Omron CX-Programmer project NewProject (CX-Programmer 9.51)

# PLC Assignment1: CP1L-E EL

## Global symbols (name address type ; comment)
1000 CHANNEL  ; O_W_E_T_Interval
T0011 BOOL  ; SRH_300

## Program NewProgram1 (cyclic task 0)
Local symbols
Arm_extends 100.05 BOOL
Arm_retracts 100.06 BOOL
Boot_Finish 2.08 BOOL  ; Has booted up
Bootup_Interval 50 NUMBER  ; Boot up for 5s
Bootup_Timer 1 NUMBER  ; Timer for bootup period
Bootup_Timer_Done T0001 BOOL  ; RUN Bootup Timer
ConvB_In_Timer 9 NUMBER  ; Timer for Conv B In
ConvB_In_Timer_Done T0009 BOOL  ; ConvB in stops
ConvB_Interval 100 NUMBER  ; ConvB stops for 10s
ConvB_Out_Interval 10.00 BOOL  ; sending pallet out for 10s
ConvB_Out_Timer 10 NUMBER  ; Timer for conv B out
ConvB_Out_Timer_Done T0010 BOOL  ; ConvB moving out timer
Converyor_B_IN 100.01 BOOL
Conveyor_A_on 100.00 BOOL
Conveyor_B_OUT 100.02 BOOL
Cycle_Count_Done C0001 BOOL  ; Cycle Counter
END_light 100.07 BOOL
EW_Mode 1.08 BOOL  ; Extend to Grab Widget Mode
End_Light_Flash_Interval 10 NUMBER  ; Flash for 1s
First_Widget 2.09 BOOL  ; if it is first widget placed
Flash_Timer1_Done T0015 BOOL  ; End Light flash 1s Timer1 ends
Flash_Timer2_Done T0016 BOOL  ; End light flash 1s Timer2 ends
GW_Interval 10 NUMBER  ; grab widget for 1s
GW_Mode 1.07 BOOL  ; Grab Widget Mode
GW_Timer 4 NUMBER  ; Timer for grab widget period
GW_Timer_Done T0004 BOOL  ; Grab Widget Timer
G_W_T_Done T0003 BOOL  ; Grip_Widget_Timer
G_W_T_Interval 50 NUMBER  ; grip widget for 5s
G_W_T_Timer 3 NUMBER  ; Timer for grip widget period
Has_Entered_Reset 2.12 BOOL  ; check if the machine has ever entered reset state
Has_Placed_Widget 2.02 BOOL  ; has placed a widet in place widget section
Has_Retract_Arm 2.05 BOOL  ; have succesfuuly retract arm to home position
LP_Mode 1.04 BOOL  ; Load pallet mode
LP_Mode_Finish 1.13 BOOL  ; load pallet mode has finished
LS1 0.03 BOOL  ; Limit Switch 1
LS2 0.04 BOOL  ; Limit Switch 2
LW_Mode 1.05 BOOL  ; Load Widget Mode
LW_Mode_Finish 1.14 BOOL  ; Load widget mode finish
MR_Interval 50 NUMBER  ; retract arm for 5s
MR_Timer 8 NUMBER  ; Timer for retract widget period
MR_Timer_Done T0008 BOOL  ; Retract After Grabbing Widget
MW_Mode 1.09 BOOL  ; Move widget mode
MW_Mode_Finish 2.01 BOOL  ; move widget mode finished
OW_Mode 1.06 BOOL  ; Obtain Widget Mode
OW_Mode_Finish 2.00 BOOL  ; Obtain Widget Mode Finished
O_W_E_T_Done T0002 BOOL  ; Obtain Widget Extend Timer
O_W_E_T_Interval 50 NUMBER  ; 5s timer
O_W_E_T_Timer 2 NUMBER  ; Timer for Obtain Widget Extend Period
Operator_present 0.07 BOOL  ; Operator present sensor
PW_Mode 1.10 BOOL  ; Place Widget Mode
PW_Mode_Finish 2.03 BOOL  ; Place Widget has finished
PW_Wait_5s T0011 BOOL  ; Forced Wait 5s according to Step 5
P_E_300_Done T0007 BOOL  ; Place Widget Extend 300 Timer
P_E_300_Interval 30 NUMBER  ; extends arm 300mm for 3s
P_E_300_Timer 7 NUMBER  ; Timer for place widget extend 300mm period
P_E_400_Done T0006 BOOL  ; Place Widget Extend 400 Timer
P_E_400_Interval 40 NUMBER  ; extends arm 400mm for 4s
P_E_400_Timer 6 NUMBER  ; Timer for place widget extend 400mm period
P_E_500_Done T0005 BOOL  ; Place Widget Extend 500 Timer
P_E_500_Interval 50 NUMBER  ; extends arm 500mm for 5s
P_E_500_Timer 5 NUMBER  ; Timer for place widget extend 500mm period
Pallet_Detected 2.07 BOOL  ; Detect pallet in Load Pallet mode
Pallet_present 0.06 BOOL  ; Pallet present sensor
Power_On 0.08 BOOL
Reset 0.02 BOOL
Reset_Interval 50 NUMBER  ; Reset pressed 5s
Reset_Mode 1.02 BOOL
Reset_Timer 0 NUMBER  ; Timer for reset period
Reset_Timer_Done T0000 BOOL  ; Reset Pressed Timer
Run_Mode 1.00 BOOL
SCARA_anticlockwise 100.04 BOOL
SCARA_clockwise 100.03 BOOL
SP_Mode 1.12 BOOL  ; Send Pallet Mode
SP_Mode_Finish 1.15 BOOL  ; Send pallet out mode finish
SRH_Mode 1.11 BOOL  ; Scara Return Home
SRH_Mode_Finish 2.04 BOOL  ; Scara Return Home has finished
SRH_R_300 T0014 BOOL  ; Retract_Arm_2_Home_3s
SRH_R_400 T0013 BOOL  ; Retract_Arm_2_Home_4s
SRH_R_500 T0012 BOOL  ; Retract_Arm_2_Home_5s
Second_Widget 2.10 BOOL  ; If it is second widget placed
Standby_Mode 1.03 BOOL
Start 0.00 BOOL
Stop 0.01 BOOL
Stop_Mode 1.01 BOOL
Stop_Mode_Finish 2.13 BOOL  ; stopped everything
Third_Widget 2.11 BOOL  ; If it is third widget placed
Vision_part_present 0.05 BOOL
Widget_Count_Done C0000 BOOL  ; Widget Counter
Widget_Count_Num 3 NUMBER  ; Number of Widgets

### Section States_Transition

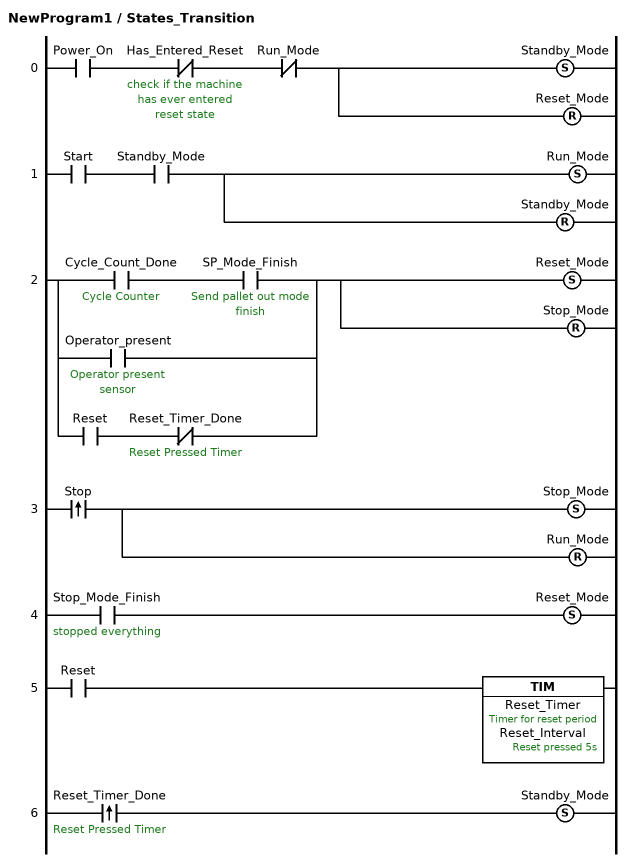
; rung 0
LD Power_On
ANDNOT Has_Entered_Reset  ; check if the machine has ever entered reset state
ANDNOT Run_Mode
SET Standby_Mode
RSET Reset_Mode
; rung 1
LD Start
AND Standby_Mode
SET Run_Mode
RSET Standby_Mode
; rung 2
LD Cycle_Count_Done  ; Cycle Counter
AND SP_Mode_Finish  ; Send pallet out mode finish
OR Operator_present  ; Operator present sensor
LD Reset
ANDNOT Reset_Timer_Done  ; Reset Pressed Timer
ORLD
SET Reset_Mode
RSET Stop_Mode
; rung 3
@LD Stop
SET Stop_Mode
RSET Run_Mode
; rung 4
LD Stop_Mode_Finish  ; stopped everything
SET Reset_Mode
; rung 5
LD Reset
TIM Reset_Timer Reset_Interval  ; Timer for reset period, Reset pressed 5s
; rung 6
@LD Reset_Timer_Done  ; Reset Pressed Timer
SET Standby_Mode

### Section Run

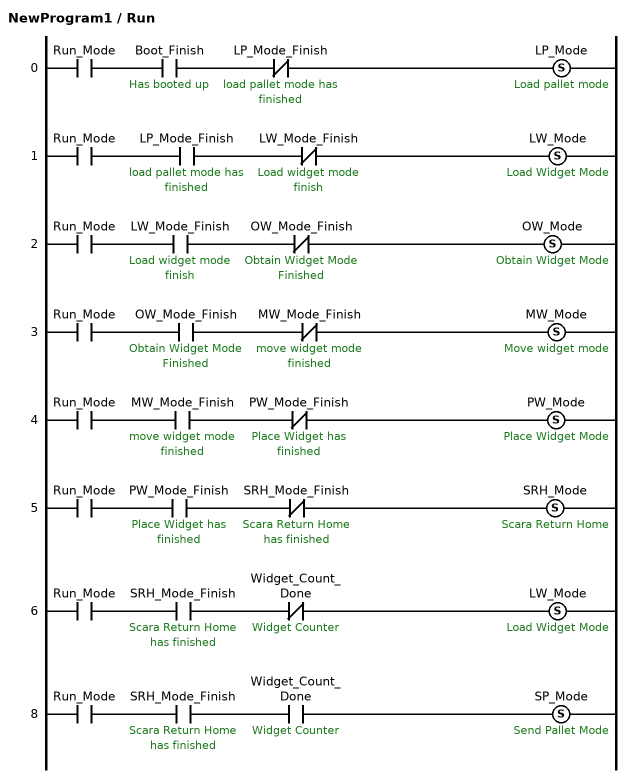
; rung 0
LD Run_Mode
AND Boot_Finish  ; Has booted up
ANDNOT LP_Mode_Finish  ; load pallet mode has finished
SET LP_Mode  ; Load pallet mode
; rung 1
LD Run_Mode
AND LP_Mode_Finish  ; load pallet mode has finished
ANDNOT LW_Mode_Finish  ; Load widget mode finish
SET LW_Mode  ; Load Widget Mode
; rung 2
LD Run_Mode
AND LW_Mode_Finish  ; Load widget mode finish
ANDNOT OW_Mode_Finish  ; Obtain Widget Mode Finished
SET OW_Mode  ; Obtain Widget Mode
; rung 3
LD Run_Mode
AND OW_Mode_Finish  ; Obtain Widget Mode Finished
ANDNOT MW_Mode_Finish  ; move widget mode finished
SET MW_Mode  ; Move widget mode
; rung 4
LD Run_Mode
AND MW_Mode_Finish  ; move widget mode finished
ANDNOT PW_Mode_Finish  ; Place Widget has finished
SET PW_Mode  ; Place Widget Mode
; rung 5
LD Run_Mode
AND PW_Mode_Finish  ; Place Widget has finished
ANDNOT SRH_Mode_Finish  ; Scara Return Home has finished
SET SRH_Mode  ; Scara Return Home
; rung 6
LD Run_Mode
AND SRH_Mode_Finish  ; Scara Return Home has finished
ANDNOT Widget_Count_Done  ; Widget Counter
SET LW_Mode  ; Load Widget Mode
; rung 8
LD Run_Mode
AND SRH_Mode_Finish  ; Scara Return Home has finished
AND Widget_Count_Done  ; Widget Counter
SET SP_Mode  ; Send Pallet Mode

### Section Stop

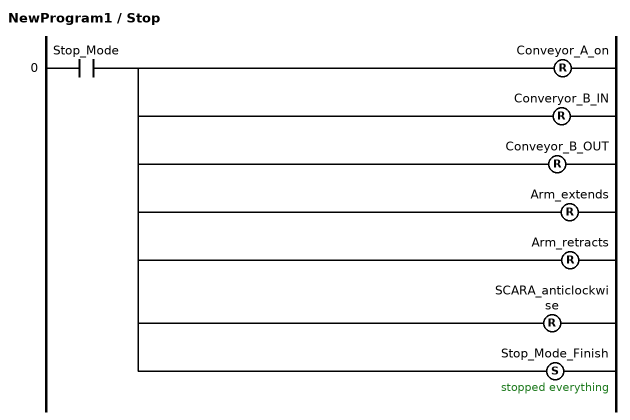
; rung 0
LD Stop_Mode
RSET Conveyor_A_on
RSET Converyor_B_IN
RSET Conveyor_B_OUT
RSET Arm_extends
RSET Arm_retracts
RSET SCARA_anticlockwise
SET Stop_Mode_Finish  ; stopped everything

### Section Reset

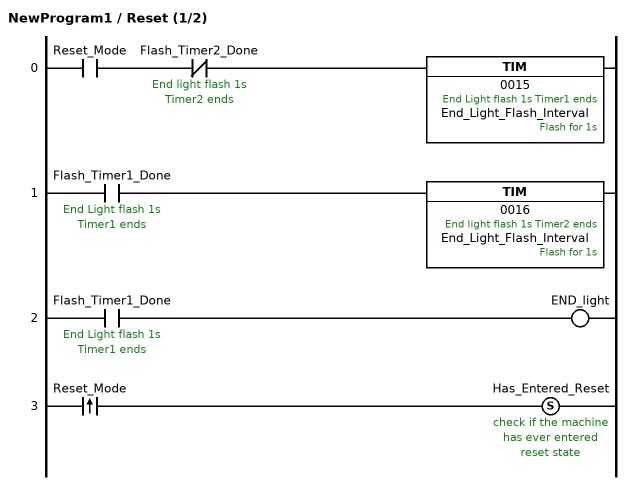
; rung 0
LD Reset_Mode
ANDNOT Flash_Timer2_Done  ; End light flash 1s Timer2 ends
TIM 0015 End_Light_Flash_Interval  ; Flash for 1s, End Light flash 1s Timer1 ends
; rung 1
LD Flash_Timer1_Done  ; End Light flash 1s Timer1 ends
TIM 0016 End_Light_Flash_Interval  ; Flash for 1s, End light flash 1s Timer2 ends
; rung 2
LD Flash_Timer1_Done  ; End Light flash 1s Timer1 ends
OUT END_light
; rung 3
@LD Reset_Mode
SET Has_Entered_Reset  ; check if the machine has ever entered reset state

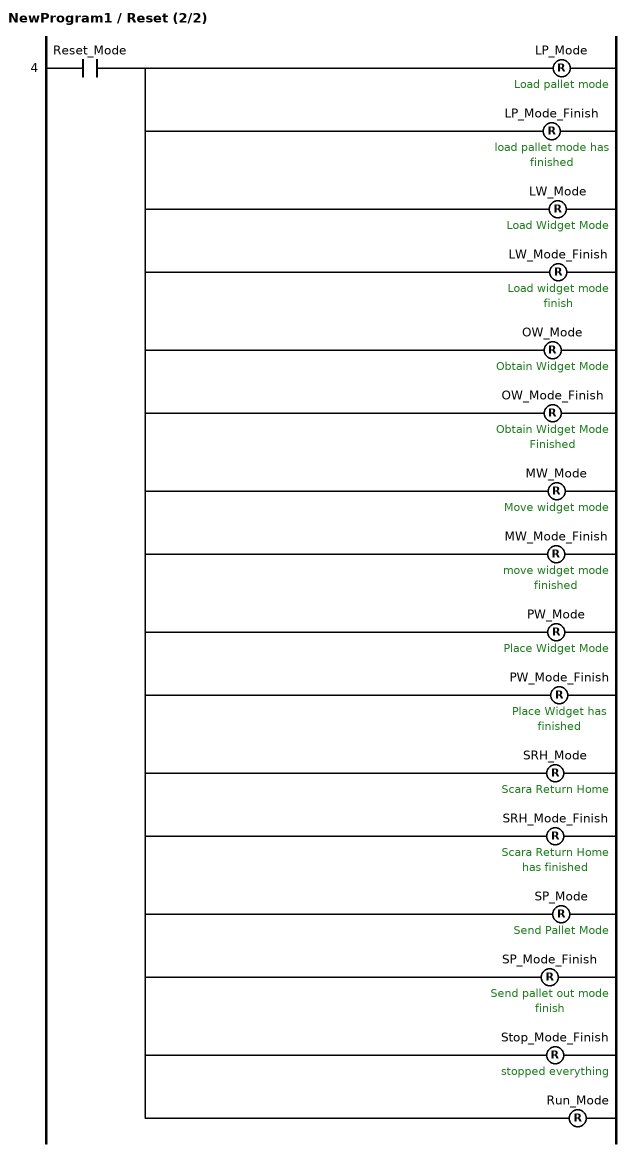
; rung 4
LD Reset_Mode
RSET LP_Mode  ; Load pallet mode
RSET LP_Mode_Finish  ; load pallet mode has finished
RSET LW_Mode  ; Load Widget Mode
RSET LW_Mode_Finish  ; Load widget mode finish
RSET OW_Mode  ; Obtain Widget Mode
RSET OW_Mode_Finish  ; Obtain Widget Mode Finished
RSET MW_Mode  ; Move widget mode
RSET MW_Mode_Finish  ; move widget mode finished
RSET PW_Mode  ; Place Widget Mode
RSET PW_Mode_Finish  ; Place Widget has finished
RSET SRH_Mode  ; Scara Return Home
RSET SRH_Mode_Finish  ; Scara Return Home has finished
RSET SP_Mode  ; Send Pallet Mode
RSET SP_Mode_Finish  ; Send pallet out mode finish
RSET Stop_Mode_Finish  ; stopped everything
RSET Run_Mode

### Section Standby

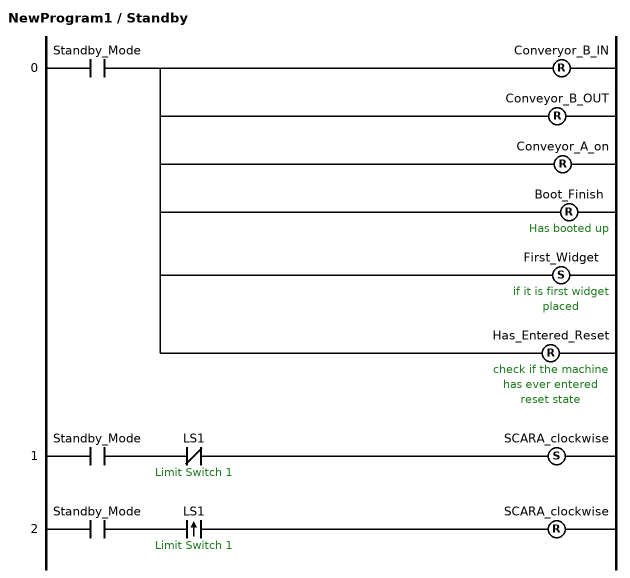
; rung 0
LD Standby_Mode
RSET Converyor_B_IN
RSET Conveyor_B_OUT
RSET Conveyor_A_on
RSET Boot_Finish  ; Has booted up
SET First_Widget  ; if it is first widget placed
RSET Has_Entered_Reset  ; check if the machine has ever entered reset state
; rung 1
LD Standby_Mode
ANDNOT LS1  ; Limit Switch 1
SET SCARA_clockwise
; rung 2
LD Standby_Mode
@AND LS1  ; Limit Switch 1
RSET SCARA_clockwise

### Section Boot_up

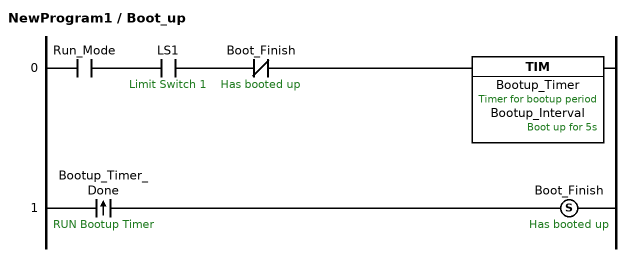
; rung 0
LD Run_Mode
AND LS1  ; Limit Switch 1
ANDNOT Boot_Finish  ; Has booted up
TIM Bootup_Timer Bootup_Interval  ; Timer for bootup period, Boot up for 5s
; rung 1
@LD Bootup_Timer_Done  ; RUN Bootup Timer
SET Boot_Finish  ; Has booted up

### Section LoadPallet

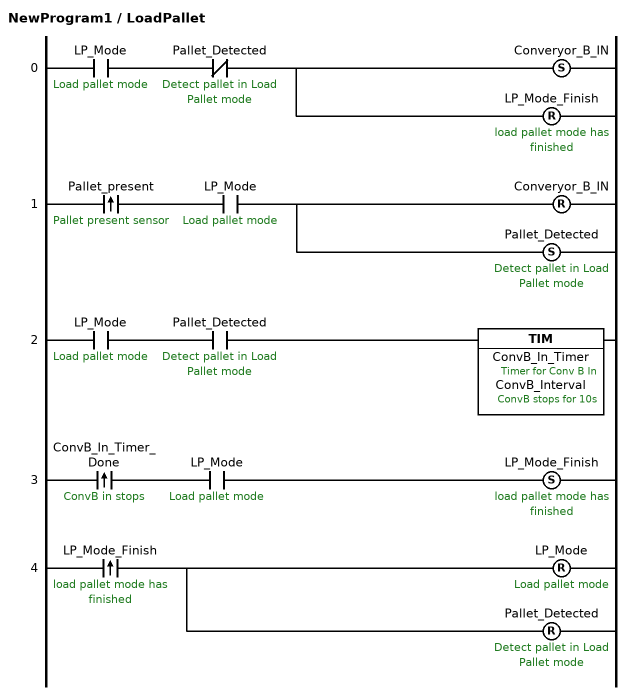
; rung 0
LD LP_Mode  ; Load pallet mode
ANDNOT Pallet_Detected  ; Detect pallet in Load Pallet mode
SET Converyor_B_IN
RSET LP_Mode_Finish  ; load pallet mode has finished
; rung 1
@LD Pallet_present  ; Pallet present sensor
AND LP_Mode  ; Load pallet mode
RSET Converyor_B_IN
SET Pallet_Detected  ; Detect pallet in Load Pallet mode
; rung 2
LD LP_Mode  ; Load pallet mode
AND Pallet_Detected  ; Detect pallet in Load Pallet mode
TIM ConvB_In_Timer ConvB_Interval  ; Timer for Conv B In, ConvB stops for 10s
; rung 3
@LD ConvB_In_Timer_Done  ; ConvB in stops
AND LP_Mode  ; Load pallet mode
SET LP_Mode_Finish  ; load pallet mode has finished
; rung 4
@LD LP_Mode_Finish  ; load pallet mode has finished
RSET LP_Mode  ; Load pallet mode
RSET Pallet_Detected  ; Detect pallet in Load Pallet mode

### Section LoadWidget

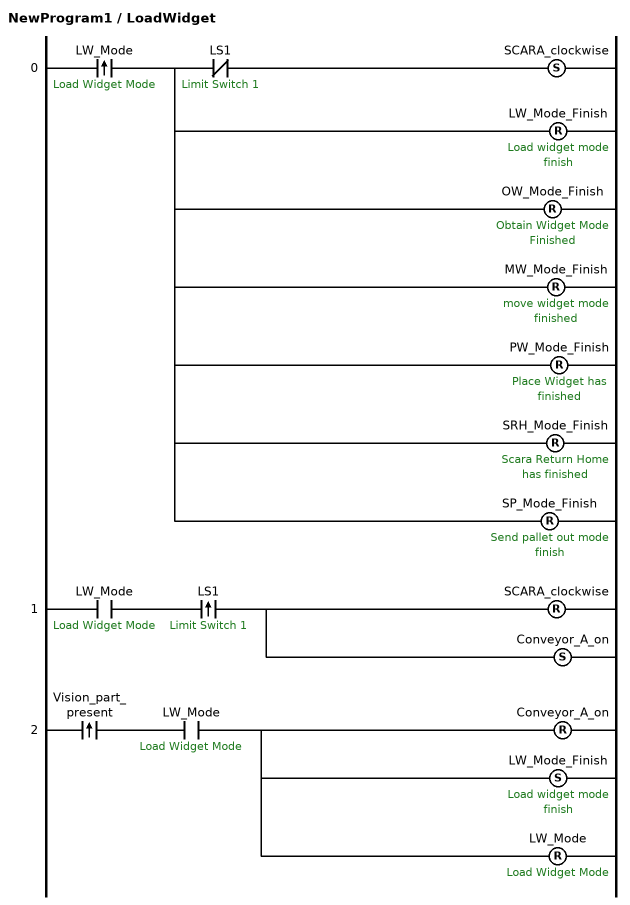
; rung 0
@LD LW_Mode  ; Load Widget Mode
OUT TR0
ANDNOT LS1  ; Limit Switch 1
SET SCARA_clockwise
LD TR0
RSET LW_Mode_Finish  ; Load widget mode finish
RSET OW_Mode_Finish  ; Obtain Widget Mode Finished
RSET MW_Mode_Finish  ; move widget mode finished
RSET PW_Mode_Finish  ; Place Widget has finished
RSET SRH_Mode_Finish  ; Scara Return Home has finished
RSET SP_Mode_Finish  ; Send pallet out mode finish
; rung 1
LD LW_Mode  ; Load Widget Mode
@AND LS1  ; Limit Switch 1
RSET SCARA_clockwise
SET Conveyor_A_on
; rung 2
@LD Vision_part_present
AND LW_Mode  ; Load Widget Mode
RSET Conveyor_A_on
SET LW_Mode_Finish  ; Load widget mode finish
RSET LW_Mode  ; Load Widget Mode

### Section ObtainWidget

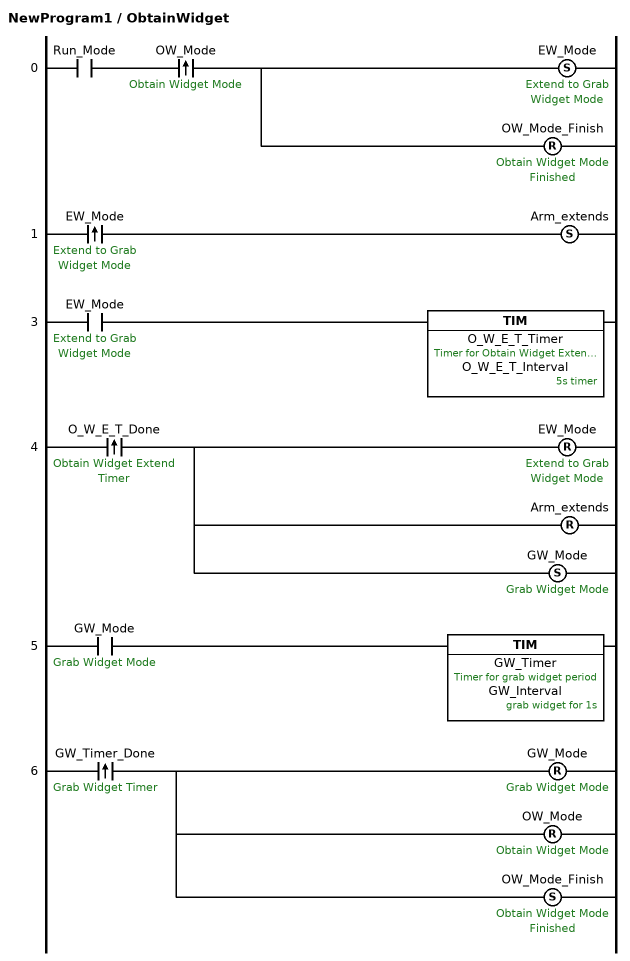
; rung 0
LD Run_Mode
@AND OW_Mode  ; Obtain Widget Mode
SET EW_Mode  ; Extend to Grab Widget Mode
RSET OW_Mode_Finish  ; Obtain Widget Mode Finished
; rung 1
@LD EW_Mode  ; Extend to Grab Widget Mode
SET Arm_extends
; rung 3
LD EW_Mode  ; Extend to Grab Widget Mode
TIM O_W_E_T_Timer O_W_E_T_Interval  ; Timer for Obtain Widget Extend Period, 5s timer
; rung 4
@LD O_W_E_T_Done  ; Obtain Widget Extend Timer
RSET EW_Mode  ; Extend to Grab Widget Mode
RSET Arm_extends
SET GW_Mode  ; Grab Widget Mode
; rung 5
LD GW_Mode  ; Grab Widget Mode
TIM GW_Timer GW_Interval  ; Timer for grab widget period, grab widget for 1s
; rung 6
@LD GW_Timer_Done  ; Grab Widget Timer
RSET GW_Mode  ; Grab Widget Mode
RSET OW_Mode  ; Obtain Widget Mode
SET OW_Mode_Finish  ; Obtain Widget Mode Finished

### Section MoveWidget

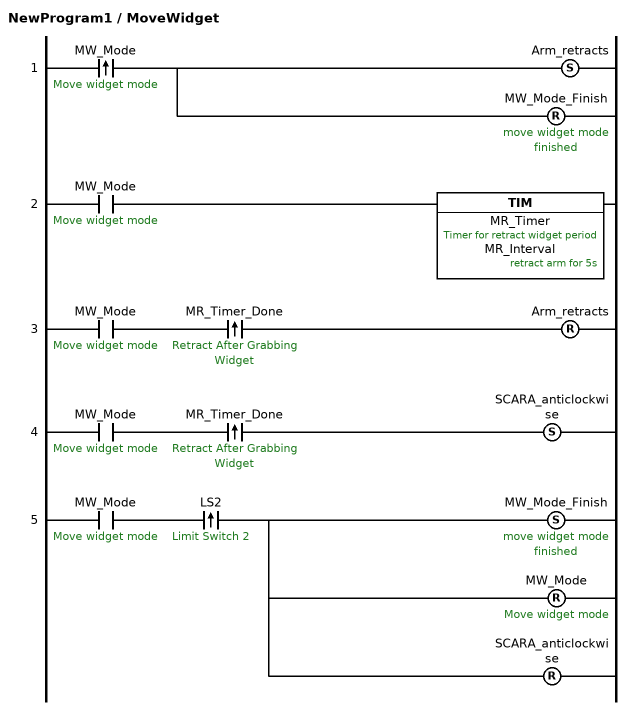
; rung 1
@LD MW_Mode  ; Move widget mode
SET Arm_retracts
RSET MW_Mode_Finish  ; move widget mode finished
; rung 2
LD MW_Mode  ; Move widget mode
TIM MR_Timer MR_Interval  ; Timer for retract widget period, retract arm for 5s
; rung 3
LD MW_Mode  ; Move widget mode
@AND MR_Timer_Done  ; Retract After Grabbing Widget
RSET Arm_retracts
; rung 4
LD MW_Mode  ; Move widget mode
@AND MR_Timer_Done  ; Retract After Grabbing Widget
SET SCARA_anticlockwise
; rung 5
LD MW_Mode  ; Move widget mode
@AND LS2  ; Limit Switch 2
SET MW_Mode_Finish  ; move widget mode finished
RSET MW_Mode  ; Move widget mode
RSET SCARA_anticlockwise

### Section PlaceWidget

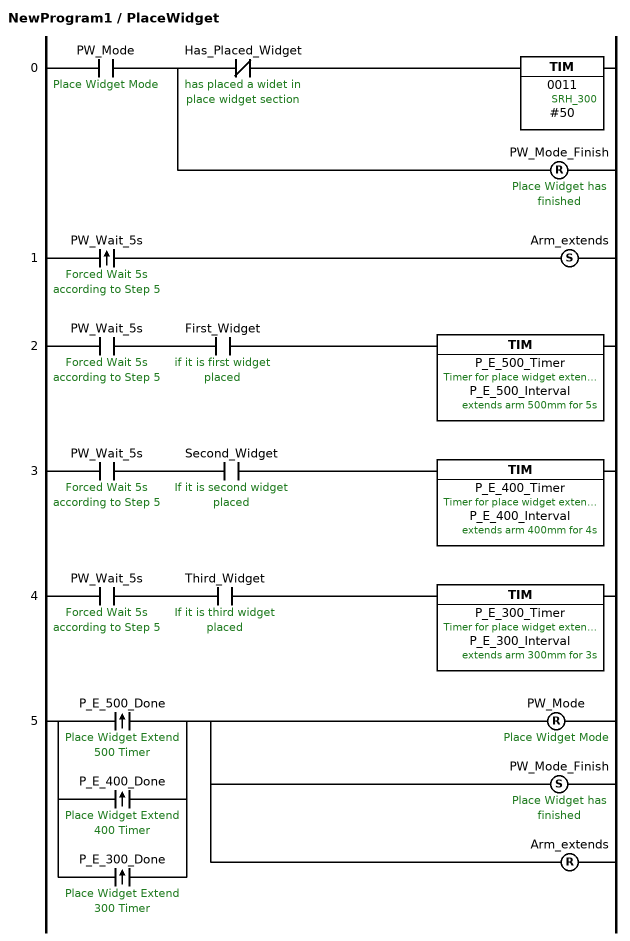
; rung 0
LD PW_Mode  ; Place Widget Mode
OUT TR0
ANDNOT Has_Placed_Widget  ; has placed a widet in place widget section
TIM 0011 #50  ; SRH_300
LD TR0
RSET PW_Mode_Finish  ; Place Widget has finished
; rung 1
@LD PW_Wait_5s  ; Forced Wait 5s according to Step 5
SET Arm_extends
; rung 2
LD PW_Wait_5s  ; Forced Wait 5s according to Step 5
AND First_Widget  ; if it is first widget placed
TIM P_E_500_Timer P_E_500_Interval  ; Timer for place widget extend 500mm period, extends arm 500mm for 5s
; rung 3
LD PW_Wait_5s  ; Forced Wait 5s according to Step 5
AND Second_Widget  ; If it is second widget placed
TIM P_E_400_Timer P_E_400_Interval  ; Timer for place widget extend 400mm period, extends arm 400mm for 4s
; rung 4
LD PW_Wait_5s  ; Forced Wait 5s according to Step 5
AND Third_Widget  ; If it is third widget placed
TIM P_E_300_Timer P_E_300_Interval  ; Timer for place widget extend 300mm period, extends arm 300mm for 3s
; rung 5
@LD P_E_500_Done  ; Place Widget Extend 500 Timer
@OR P_E_400_Done  ; Place Widget Extend 400 Timer
@OR P_E_300_Done  ; Place Widget Extend 300 Timer
RSET PW_Mode  ; Place Widget Mode
SET PW_Mode_Finish  ; Place Widget has finished
RSET Arm_extends

### Section ScaraReturnHome

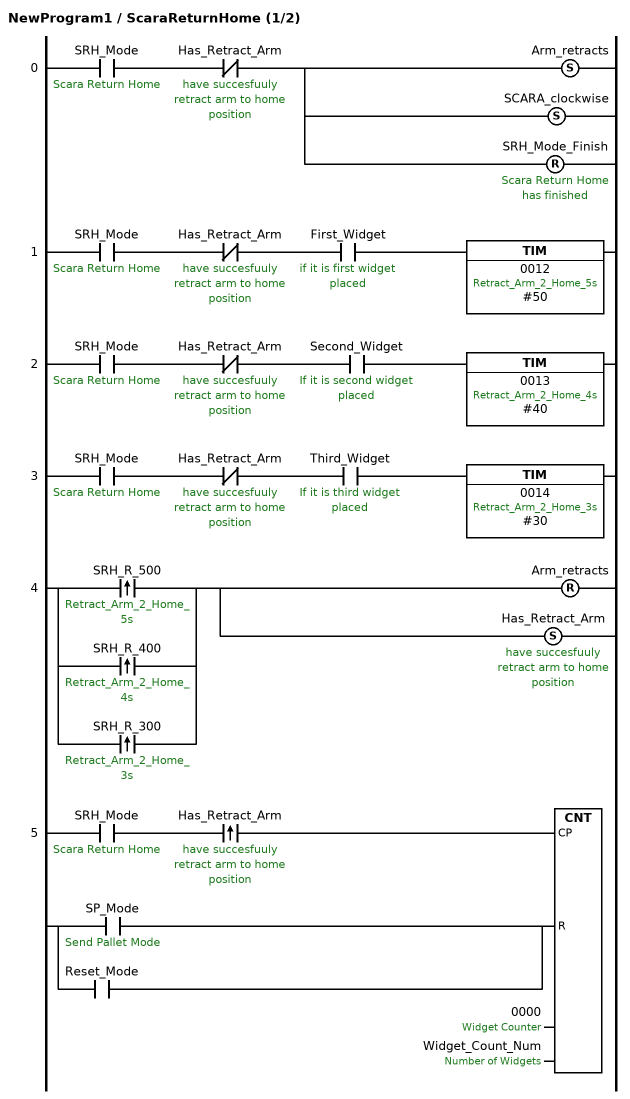
; rung 0
LD SRH_Mode  ; Scara Return Home
ANDNOT Has_Retract_Arm  ; have succesfuuly retract arm to home position
SET Arm_retracts
SET SCARA_clockwise
RSET SRH_Mode_Finish  ; Scara Return Home has finished
; rung 1
LD SRH_Mode  ; Scara Return Home
ANDNOT Has_Retract_Arm  ; have succesfuuly retract arm to home position
AND First_Widget  ; if it is first widget placed
TIM 0012 #50  ; Retract_Arm_2_Home_5s
; rung 2
LD SRH_Mode  ; Scara Return Home
ANDNOT Has_Retract_Arm  ; have succesfuuly retract arm to home position
AND Second_Widget  ; If it is second widget placed
TIM 0013 #40  ; Retract_Arm_2_Home_4s
; rung 3
LD SRH_Mode  ; Scara Return Home
ANDNOT Has_Retract_Arm  ; have succesfuuly retract arm to home position
AND Third_Widget  ; If it is third widget placed
TIM 0014 #30  ; Retract_Arm_2_Home_3s
; rung 4
@LD SRH_R_500  ; Retract_Arm_2_Home_5s
@OR SRH_R_400  ; Retract_Arm_2_Home_4s
@OR SRH_R_300  ; Retract_Arm_2_Home_3s
RSET Arm_retracts
SET Has_Retract_Arm  ; have succesfuuly retract arm to home position
; rung 5
LD SRH_Mode  ; Scara Return Home
@AND Has_Retract_Arm  ; have succesfuuly retract arm to home position
LD SP_Mode  ; Send Pallet Mode
OR Reset_Mode
CNT 0000 Widget_Count_Num  ; Number of Widgets, Widget Counter

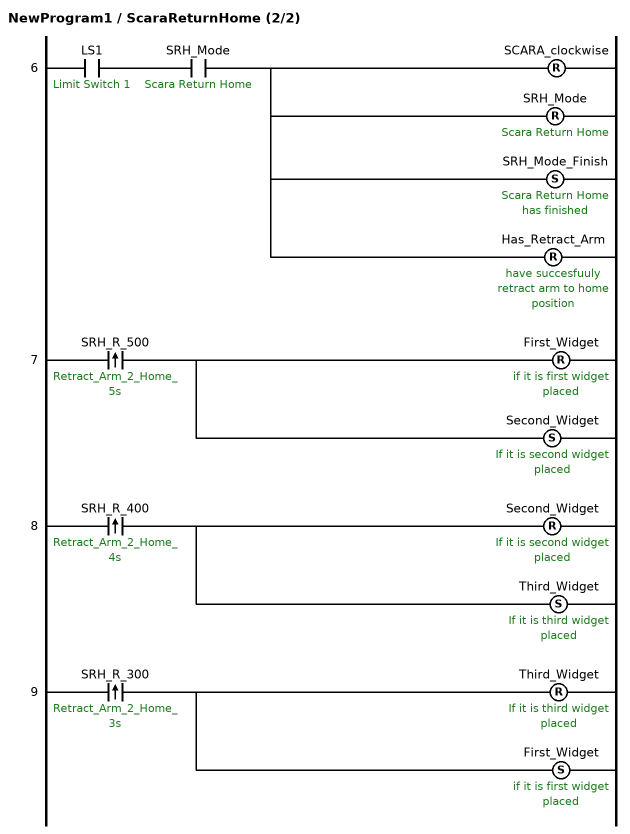
; rung 6
LD LS1  ; Limit Switch 1
AND SRH_Mode  ; Scara Return Home
RSET SCARA_clockwise
RSET SRH_Mode  ; Scara Return Home
SET SRH_Mode_Finish  ; Scara Return Home has finished
RSET Has_Retract_Arm  ; have succesfuuly retract arm to home position
; rung 7
@LD SRH_R_500  ; Retract_Arm_2_Home_5s
RSET First_Widget  ; if it is first widget placed
SET Second_Widget  ; If it is second widget placed
; rung 8
@LD SRH_R_400  ; Retract_Arm_2_Home_4s
RSET Second_Widget  ; If it is second widget placed
SET Third_Widget  ; If it is third widget placed
; rung 9
@LD SRH_R_300  ; Retract_Arm_2_Home_3s
RSET Third_Widget  ; If it is third widget placed
SET First_Widget  ; if it is first widget placed

### Section SendPallet

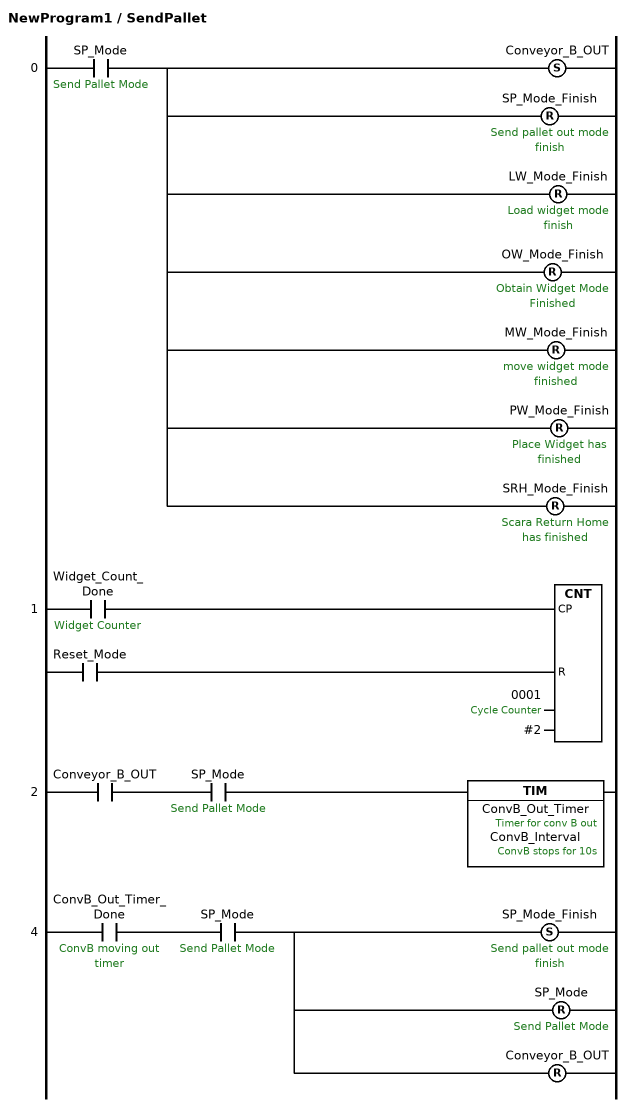
; rung 0
LD SP_Mode  ; Send Pallet Mode
SET Conveyor_B_OUT
RSET SP_Mode_Finish  ; Send pallet out mode finish
RSET LW_Mode_Finish  ; Load widget mode finish
RSET OW_Mode_Finish  ; Obtain Widget Mode Finished
RSET MW_Mode_Finish  ; move widget mode finished
RSET PW_Mode_Finish  ; Place Widget has finished
RSET SRH_Mode_Finish  ; Scara Return Home has finished
; rung 1
LD Widget_Count_Done  ; Widget Counter
LD Reset_Mode
CNT 0001 #2  ; Cycle Counter
; rung 2
LD Conveyor_B_OUT
AND SP_Mode  ; Send Pallet Mode
TIM ConvB_Out_Timer ConvB_Interval  ; Timer for conv B out, ConvB stops for 10s
; rung 4
LD ConvB_Out_Timer_Done  ; ConvB moving out timer
AND SP_Mode  ; Send Pallet Mode
SET SP_Mode_Finish  ; Send pallet out mode finish
RSET SP_Mode  ; Send Pallet Mode
RSET Conveyor_B_OUT

### Section END
; rung 0
END(001)